(* PLC project SafeLOGIC-1, BrAutomation SafeDESIGNER  4.3.0.6 *)
(* stored: companyURL http://www.br-automation.com, creationDateTime Wed Aug 16 14:59:49 2017 *)

PROGRAM Main

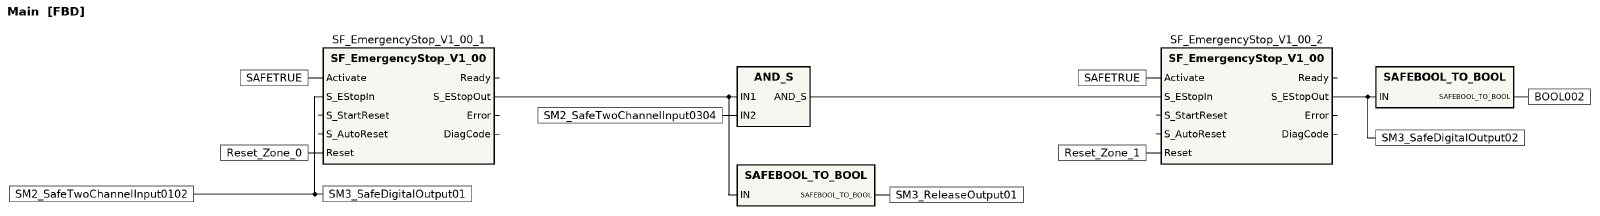
(* FBD diagram, written out as Structured Text *)
SM3_SafeDigitalOutput01 := SM2_SafeTwoChannelInput0102;
SF_EmergencyStop_V1_00_1(Activate := SAFETRUE, S_EStopIn := SM2_SafeTwoChannelInput0102, Reset := Reset_Zone_0);
SM3_ReleaseOutput01 := SAFEBOOL_TO_BOOL(SF_EmergencyStop_V1_00_1.S_EStopOut);
SF_EmergencyStop_V1_00_2(Activate := SAFETRUE, S_EStopIn := AND_S(SF_EmergencyStop_V1_00_1.S_EStopOut, SM2_SafeTwoChannelInput0304), Reset := Reset_Zone_1);
SM3_SafeDigitalOutput02 := SF_EmergencyStop_V1_00_2.S_EStopOut;
BOOL002 := SAFEBOOL_TO_BOOL(SF_EmergencyStop_V1_00_2.S_EStopOut);
END_PROGRAM
